FUNCTION_BLOCK FB_ErrorSystem

VAR_INPUT
	En					: BOOL;							//Enable input
	bReset				: BOOL;							//Delete all Error entry
	nErrorID			: ULINT;						//ErrorID to be acknoledged
	bACK				: BOOL;							//Acknoledge the given error and delete it from the list
	bValidSelection		: BOOL;							//Visu table valid selection flag
	nTableRowIndex		: INT;							//Visu table selected row index
END_VAR
	
VAR_OUTPUT
	EnO 				: BOOL;							//Enable output
	nSelectedError		: ULINT;						//Currently selected errorID
	nNoError			: UINT;							//Number of Errors
	nActive				: UINT;							//Number of Active Errors
	nInactive			: UINT;							//Number of Inactive Errors
	nNoOverflow			: INT;							//Number of Overflows
	pErrorSystem 		: POINTER TO ST_ErrorSystem;	//Pointer to ErrorSystem
END_VAR

VAR_IN_OUT
	
END_VAR

VAR
	nFreePos : UINT;									//Number of free position in the list
	nListCnt1 : UINT;									//work variable
	ErrorSystem : ST_ErrorSystem;						//Data structure of the Error list
	
	bAckInternal		: BOOL;
	bResetInternal		: BOOL;
	nErrorIDInternal	: ULINT;
	
	Ack_trig		: R_TRIG;
	RST_trig		: R_TRIG;
END_VAR

(*
* ================================================================================
*                                   DESCRIPTION
* ================================================================================
* This Function Block implements the core structure of the Error/Warning Handling
* system. It realizes the datastructure containing every Error Entry, collect
* statistics about the usage and manage the Error Entries.
* ================================================================================
*)
EnO := En;

//Ponter to ErrorSystem
pErrorSystem := ADR(ErrorSystem);

//Number of overflows
nNoOverflow := ErrorSystem.nNoOverflows;

Ack_trig (
	CLK		:= bAck,
	Q		=> bAckInternal,
);

RST_trig (
	CLK		:= bReset,
	Q		=> bResetInternal,
);

IF bValidSelection AND nErrorID = 0 THEN
	nErrorIDInternal := ErrorSystem.aErrorData[nTableRowIndex].Error_ID;
ELSE
	nErrorIDInternal := nErrorID;
END_IF

nSelectedError := nErrorIDInternal;

IF bResetInternal THEN
	MEMSET ( ADR(ErrorSystem.aErrorData[0]), 0, cSizeOfErrorData * SIZEOF(ST_ErrorEntry));
	ErrorSystem.nNextErrorID := 1;
END_IF

//Number of errors in the system
nNoError := 0;
nActive := 0;
nInactive := 0;
FOR nListCnt1 := 0 TO cSizeOfErrorData - 1 DO
	IF ErrorSystem.aErrorData[nListCnt1].Error_ID <> 0  THEN
		nNoError := nNoError+1;
		IF ErrorSystem.aErrorData[nListCnt1].ErrorState = DUT_ErrorState.Active THEN
			nActive := nActive + 1;
		ELSE
			nInactive := nInactive + 1;
		END_IF
	END_IF
END_FOR
ErrorSystem.nNoErrors := nNoError;

//Number of free position in the list
nFreePos := cSizeOfErrorData - nNoError;

//Acknoledge specified Error entry
IF bAckInternal THEN
	FOR nListCnt1 := 0 TO cSizeOfErrorData - 1 DO
		IF ErrorSystem.aErrorData[nListCnt1].Error_ID = nErrorIDInternal THEN
			ErrorSystem.aErrorData[nListCnt1].ErrorState := DUT_ErrorState.Acknowledged;
		END_IF
	END_FOR
END_IF

//Deleting acknoledged errors
FOR nListCnt1 := 0 TO cSizeOfErrorData - 1 DO
	IF ErrorSystem.aErrorData[nListCnt1].ErrorState = DUT_ErrorState.Acknowledged THEN
		MEMMOVE (ADR(ErrorSystem.aErrorData[nListCnt1]), ADR(ErrorSystem.aErrorData[nListCnt1+1]), (cSizeOfErrorData - 1 - nListCnt1) * SIZEOF(ST_ErrorEntry));
		MEMSET(ADR(ErrorSystem.aErrorData[cSizeOfErrorData - 1]), 0, SIZEOF(ST_ErrorEntry));
	END_IF
END_FOR

END_FUNCTION_BLOCK

(* stored: Version 1.1.0.1, ProductVersion 3.1.4022.17
   POU FB_ErrorSystem: Id {978ea49f-a940-4b4e-9f45-8cdde4adcf37}, SpecialFunc None *)
